// TIA Portal V20 export
TYPE "LDrive_typeKistlerParameters"
// stored: IsFailsafeCompliant false
   STRUCT
      UNI_in { ExternalAccessible := 'False'; ExternalVisible := 'False'; ExternalWritable := 'False'} : Array[0..7] of Bool;
      universalvariables { ExternalAccessible := 'False'; ExternalVisible := 'False'; ExternalWritable := 'False'} : Array[0..9] of Real;
   END_STRUCT;
END_TYPE
